{attribute 'linkalways'} 
{attribute 'no_explicit_call' := 'This FB is a CLASS and must be accessed using methods or properties'}
{attribute 'enable_dynamic_creation'}
FUNCTION_BLOCK Node_F_VN_HistogramEqualization EXTENDS VisionNode
VAR
	ipSrcImage : _ITcVnImage;
    ipDestImage : _ITcVnImage;
    hrPrev : _HRESULT(S_OK);
	hresult : _HRESULT(S_OK);
END_VAR

METHOD PUBLIC  Clone : I_Node
VAR
	pNode : POINTER TO Node_F_VN_HistogramEqualization;
END_VAR
pNode := __NEW(Node_F_VN_HistogramEqualization);
Clone := pNode^;
END_METHOD

METHOD FB_init : BOOL
VAR_INPUT
	bInitRetains : BOOL; // if TRUE, the retain variables are initialized (warm start / cold start)
	bInCopyCode : BOOL;  // if TRUE, the instance afterwards gets moved into the copy code (online change)
END_VAR
AddInput('ipSrcImage', ipSrcImage);
AddInput('hrPrev', hrPrev);
AddOutput('ipDestImage', ipDestImage);
AddOutput('hresult',hresult);
END_METHOD

METHOD PROTECTED OnExecute
hresult.Value := F_VN_HistogramEqualization(
	ipSrcImage   := ipSrcImage.Value,
    ipDestImage   := ipDestImage.Value,
	hrPrev := hrPrev.Value);
END_METHOD

METHOD PUBLIC PreExecutionCheck
VAR_INPUT
	Check : I_PreExecutionChecks;
END_VAR
Check.IsTrue(ipSrcImage.IsValid, 'ipSrcImage must contain an image');
Check.IsTrue((ipSrcImage.HasChannelCount(1) OR ipSrcImage.HasChannelCount(3)), 'ipSrcImage must have 1 or 3 channels');
END_METHOD

END_FUNCTION_BLOCK

(* stored: Version 1.1.0.1, ProductVersion 3.1.4024.13
   POU Node_F_VN_HistogramEqualization: Id {e5494efa-6075-0d37-28e3-5d232a6a50fc}, SpecialFunc None
   Folder Constructor: Id {f0b1aa67-865e-0632-2a70-cef295d64c0a}
   Method Clone: Id {19001e92-ea4d-004e-09ba-38b3f636fdb8}
   Method FB_init: Id {7814c119-0a90-0caa-0776-cae2621dfaac}
   Method OnExecute: Id {3c9ecc22-916f-0d55-2d93-e931f1fa45e8}
   Method PreExecutionCheck: Id {f968c360-b3c4-01b0-2097-1297e92edace} *)
